{attribute 'qualified_only'}
VAR_GLOBAL CONSTANT
	MaxMessages : USINT := 10;
END_VAR

(* stored: Version 1.1.0.1, ProductVersion 3.1.4026.18
   GVL Parameters: Id {99125352-013f-4f7e-9fb1-ea9b5af710a7}, ParameterList True *)
